FUNCTION_BLOCK FB_Bel_Ablaufsteuerung
VAR_IN_OUT
	Zustand			: ST_Bel_Zustand;
	Stellwert		: ST_Bel_Stellwert;
END_VAR
VAR_INPUT
	Steuerung		: ST_Bel_Steuerung;
	Parameter		: ST_Bel_Parameter;
END_VAR
VAR_OUTPUT
END_VAR
VAR
	Timer: TON;
END_VAR

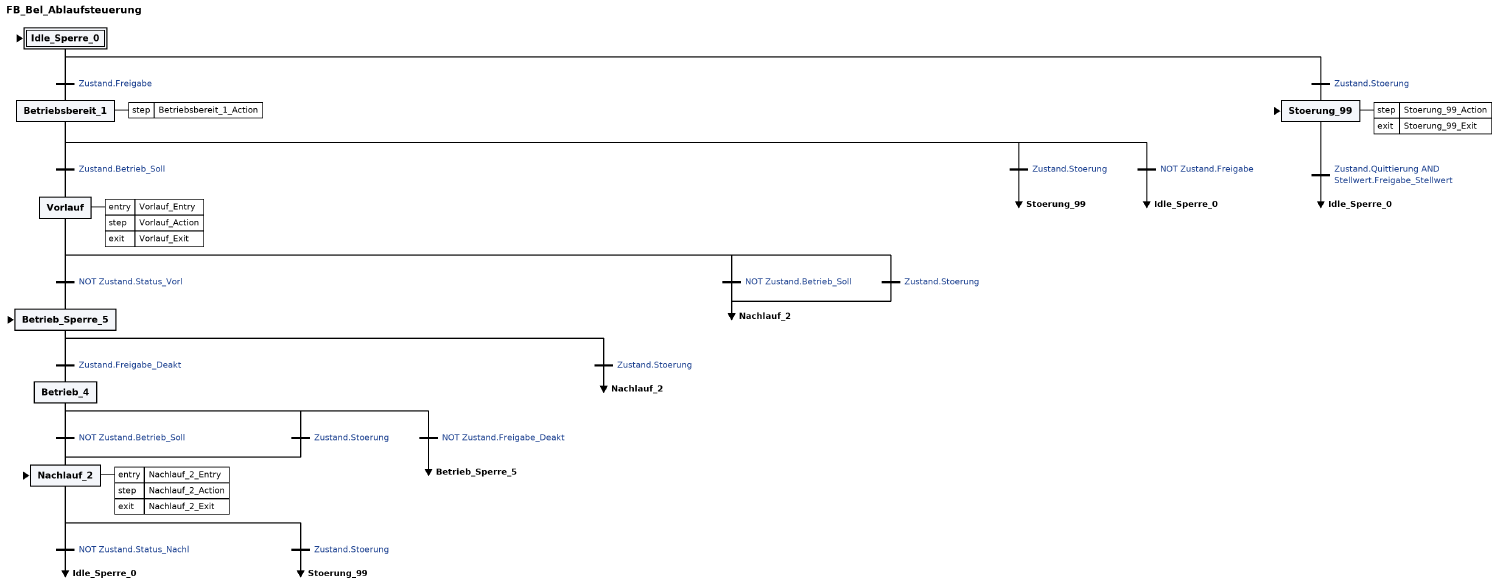
INITIAL_STEP Idle_Sperre_0:
END_STEP
TRANSITION FROM Idle_Sperre_0 TO Betriebsbereit_1
    := Zustand.Freigabe;
END_TRANSITION
TRANSITION FROM Idle_Sperre_0 TO Stoerung_99
    := Zustand.Stoerung;
END_TRANSITION
STEP Stoerung_99:
    Stoerung_99_Action(N);  // step action
    Stoerung_99_Exit(P0);  // exit action
END_STEP
TRANSITION FROM Stoerung_99 TO Idle_Sperre_0
    := Zustand.Quittierung AND Stellwert.Freigabe_Stellwert;
END_TRANSITION
STEP Betriebsbereit_1:
    Betriebsbereit_1_Action(N);  // step action
END_STEP
TRANSITION FROM Betriebsbereit_1 TO Vorlauf
    := Zustand.Betrieb_Soll;
END_TRANSITION
TRANSITION FROM Betriebsbereit_1 TO Stoerung_99
    := Zustand.Stoerung;
END_TRANSITION
TRANSITION FROM Betriebsbereit_1 TO Idle_Sperre_0
    := NOT Zustand.Freigabe;
END_TRANSITION
STEP Vorlauf:
    Vorlauf_Entry(P1);  // entry action
    Vorlauf_Action(N);  // step action
    Vorlauf_Exit(P0);  // exit action
END_STEP
TRANSITION FROM Vorlauf TO Betrieb_Sperre_5
    := NOT Zustand.Status_Vorl;
END_TRANSITION
TRANSITION FROM Vorlauf TO Nachlauf_2
    := NOT Zustand.Betrieb_Soll;
END_TRANSITION
TRANSITION FROM Vorlauf TO Nachlauf_2
    := Zustand.Stoerung;
END_TRANSITION
STEP Betrieb_Sperre_5:
END_STEP
TRANSITION FROM Betrieb_Sperre_5 TO Betrieb_4
    := Zustand.Freigabe_Deakt;
END_TRANSITION
TRANSITION FROM Betrieb_Sperre_5 TO Nachlauf_2
    := Zustand.Stoerung;
END_TRANSITION
STEP Betrieb_4:
END_STEP
TRANSITION FROM Betrieb_4 TO Nachlauf_2
    := NOT Zustand.Betrieb_Soll;
END_TRANSITION
TRANSITION FROM Betrieb_4 TO Nachlauf_2
    := Zustand.Stoerung;
END_TRANSITION
TRANSITION FROM Betrieb_4 TO Betrieb_Sperre_5
    := NOT Zustand.Freigabe_Deakt;
END_TRANSITION
STEP Nachlauf_2:
    Nachlauf_2_Entry(P1);  // entry action
    Nachlauf_2_Action(N);  // step action
    Nachlauf_2_Exit(P0);  // exit action
END_STEP
TRANSITION FROM Nachlauf_2 TO Idle_Sperre_0
    := NOT Zustand.Status_Nachl;
END_TRANSITION
TRANSITION FROM Nachlauf_2 TO Stoerung_99
    := Zustand.Stoerung;
END_TRANSITION

ACTION Betriebsbereit_1_Action:
Stellwert.Freigabe_Stellwert := TRUE;
END_ACTION

ACTION Nachlauf_2_Action:
(* Nachlauf Timer starten *)
Timer( 	IN := Zustand.Status_Nachl,
		PT := DINT_TO_TIME(Parameter.Zeit_Nachl)
);
Zustand.Status_Nachl	:= NOT(Timer.Q AND NOT Zustand.Betrieb);

(* Stellwert setzen *)
Stellwert.Betrieb := FALSE;
Stellwert.Freigabe_Stellwert := FALSE;

(* Zustand setzen *)
Zustand.Status := E_Bel_Zustand_Status_Nachl;
END_ACTION

ACTION Nachlauf_2_Entry:
Zustand.Status_Nachl := TRUE;
(* Reset Timer *)
Timer(IN := FALSE);
END_ACTION

ACTION Nachlauf_2_Exit:
Zustand.Status_Nachl := FALSE;
END_ACTION

ACTION Stoerung_99_Action:
(* Stellwert setzen *)
Stellwert.Betrieb := FALSE;

(* Zustand setzen *)
Zustand.Stoerung := TRUE;
Zustand.Status := E_Bel_Zustand_Status_Stoerung;
END_ACTION

ACTION Stoerung_99_Exit:
Zustand.Stoerung	:= FALSE;
END_ACTION

ACTION Vorlauf_Action:
(* Vorlaufzeit Timer starten *)
Timer( 	IN := Zustand.Status_Vorl,
		PT := DINT_TO_TIME(Parameter.Zeit_Vorl)
);
Zustand.Status_Vorl := NOT (Timer.Q AND Zustand.Betrieb);

(* Stellwert setzen *)
IF Stellwert.Freigabe_Stellwert = TRUE THEN
	Stellwert.Betrieb := TRUE;
END_IF

(* Zustand setzen *)
Zustand.Status := E_Bel_Zustand_Status_Vorl;
END_ACTION

ACTION Vorlauf_Entry:
Zustand.Status_Vorl := TRUE;
(* Reset Timer *)
Timer(IN := FALSE);
END_ACTION

ACTION Vorlauf_Exit:
Zustand.Status_Vorl := FALSE;
END_ACTION

END_FUNCTION_BLOCK

(* stored: Version 1.1.0.1, ProductVersion 3.1.4024.10
   POU FB_Bel_Ablaufsteuerung: Id {6a49ac82-cd62-4f98-89ce-d1001bf0ed23}, SpecialFunc None
   Action Betriebsbereit_1_Action: Id {e291c243-623c-4c37-a980-161e6759d8f6}
   Action Nachlauf_2_Action: Id {671526f7-50ed-4183-a6a5-a4a606c19646}
   Action Nachlauf_2_Entry: Id {f807e387-79fe-432c-9242-bb1e85d42a13}
   Action Nachlauf_2_Exit: Id {247c4cf3-b98e-4ffc-bae8-03bbcf85d74e}
   Action Stoerung_99_Action: Id {d9e5db17-48e6-4ee3-887b-43de38d94117}
   Action Stoerung_99_Exit: Id {078f1318-fef6-4b39-88e6-34fd2b7654c8}
   Action Vorlauf_Action: Id {7fff6f07-96ed-468b-bc89-47fd2506e9d4}
   Action Vorlauf_Entry: Id {aa951045-d8d0-451c-a0aa-5d5edeb85bf4}
   Action Vorlauf_Exit: Id {b7b149dd-7000-420f-a579-c41c9d1168c0} *)
